{attribute addProperty BoxType "EL6201-0000-0017"}
{attribute addProperty Id "Slave_13A_DO0BIT10.12597Slave_13A_DO1BIT10.12598Slave_13A_DO2BIT10.12599Slave_13A_DO3BIT10.125100Slave_13B_DO0BIT10.125101Slave_13B_DO1BIT10.125102Slave_13B_DO2BIT10.125103Slave_13B_DO3BIT10.125104"}
{attribute addProperty CRC "3588165749"}
{attribute addProperty SizeInBites "8"}
{attribute addProperty SizeInBytes "1"}
TYPE Slave_13_Outputs_D5DF1075 :
STRUCT
	{attribute addProperty Name "Slave_13A_DO0"}
	Slave_13A_DO0 : BIT;
	{attribute addProperty Name "Slave_13A_DO1"}
	Slave_13A_DO1 : BIT;
	{attribute addProperty Name "Slave_13A_DO2"}
	Slave_13A_DO2 : BIT;
	{attribute addProperty Name "Slave_13A_DO3"}
	Slave_13A_DO3 : BIT;
	{attribute addProperty Name "Slave_13B_DO0"}
	Slave_13B_DO0 : BIT;
	{attribute addProperty Name "Slave_13B_DO1"}
	Slave_13B_DO1 : BIT;
	{attribute addProperty Name "Slave_13B_DO2"}
	Slave_13B_DO2 : BIT;
	{attribute addProperty Name "Slave_13B_DO3"}
	Slave_13B_DO3 : BIT;
END_STRUCT
END_TYPE

(* stored: Version 1.2.0.0, ProductVersion 3.1.4024.9
   DUT Slave_13_Outputs_D5DF1075: Id {3bcfd320-ec04-4ef1-8d44-b453c50cd04b} *)
